ABB RobotStudio station: conveyor SS.rsstn

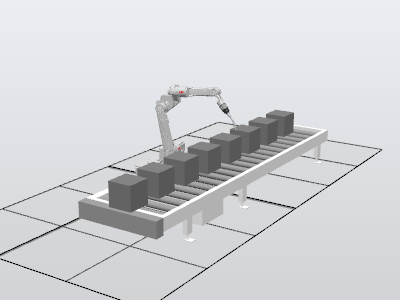
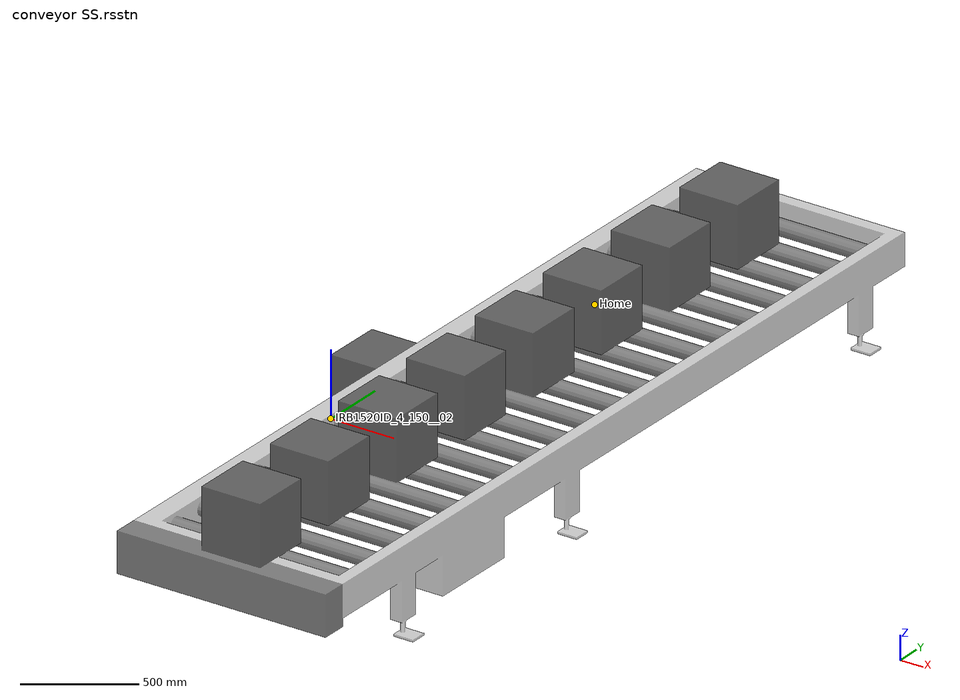
[picture v1: parts stored in the station drawn from their meshes, with robot base, taught points and paths (robot models come from the ABB library and are not in the file)]
Station Station (saved by RobotStudio 22.3.10141.1)
Controller Controller51, task T_ROB1: task frame (RAPID world) sits at (490, 760, 435) mm, rotated rx 0 ry 0 rz -90 deg in the station
Controller Controller51
  mechanical unit ROB_1: IRB1520ID_4_150__02, 6 joints, base frame (760, -490, -435) mm, rotated rx 0 ry 0 rz 90 deg
  mechanical unit CNV1: ?, 1 joints, base frame (0, 0, 0) mm
Layout (positions relative to the parent item):
  - IRB1520ID_4_150__02 [mechanism] at (0, 0, 0) mm; joint values [0.1337, -0.205, 0.1243, -0.1103, 0.9334, 0.1661] (rad or m)
      links: Base, Link1, Link2, Link3, Link4, Link5, Link6
  - Binzel_ID_22 [mechanism, from Tools\Binzel_ID_22.rslib] at (870.51, 99.26, 1138.57) mm, rotated rx 180 ry 41.56 rz 180 deg
  - Conveyor [conveyor]
    - 950_4000_h2 [part] at (1400, -2000, 0) mm, rotated rx 0 ry 0 rz 90 deg, size 4244 x 1170 x 435 mm
    - Box [part], size 300 x 300 x 300 mm
    - ConveyorObject_1 [conveyorobject] at (490, -1725.53, 435) mm, rotated rx 0 ry 0 rz -90 deg
      - Box [part] at (50, 300, 0) mm, size 300 x 300 x 300 mm
    - ConveyorObject_2 [conveyorobject] at (490, -1225.53, 435) mm, rotated rx 0 ry 0 rz -90 deg
      - Box [part] at (50, 300, 0) mm, size 300 x 300 x 300 mm
    - ConveyorObject_3 [conveyorobject] at (490, -725.53, 435) mm, rotated rx 0 ry 0 rz -90 deg
      - Box [part] at (50, 300, 0) mm, size 300 x 300 x 300 mm
    - ConveyorObject_4 [conveyorobject] at (490, -225.53, 435) mm, rotated rx 0 ry 0 rz -90 deg
      - Box [part] at (50, 300, 0) mm, size 300 x 300 x 300 mm
    - ConveyorObject_5 [conveyorobject] at (490, 274.47, 435) mm, rotated rx 0 ry 0 rz -90 deg
      - Box [part] at (50, 300, 0) mm, size 300 x 300 x 300 mm
    - ConveyorObject_6 [conveyorobject] at (490, 774.47, 435) mm, rotated rx 0 ry 0 rz -90 deg
      - Box [part] at (50, 300, 0) mm, size 300 x 300 x 300 mm
    - ConveyorObject_7 [conveyorobject] at (490, 1274.47, 435) mm, rotated rx 0 ry 0 rz -90 deg
      - Box [part] at (50, 300, 0) mm, size 300 x 300 x 300 mm
    - ConveyorObject_8 [conveyorobject] at (490, 1774.47, 435) mm, rotated rx 0 ry 0 rz -90 deg
      - Box [part] at (50, 300, 0) mm, size 300 x 300 x 300 mm
Attachment: Binzel_ID_22 is attached to IRB1520ID_4_150__02 / Link6
Conveyor tracking Connection_4: unit CNV1, TravelOffset=1.3, QueueTrackDistance=0, StartWindowWidth=1.5, SyncSeparation=0, CountsPerMeter=10000
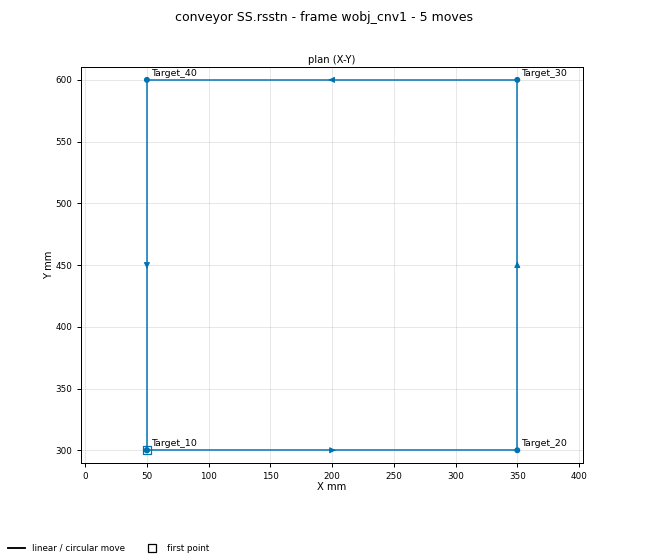
[picture p0: tool path of conveyor SS.rsstn in frame wobj_cnv1, 5 of 7 moves have a stored position in this frame; points joined in program order, loops and branches not executed]
Targets, tools, work objects and paths stored in the station, written as RAPID:
! task T_ROB1
MODULE CalibData
  PERS tooldata tWeldGun:=[TRUE,[[49.841566361,0,372.194826196],[0.981627183,0,0.190808995,0]],[2,[0,0,100],[0,1,0,0],0,0,0]];
  TASK PERS wobjdata wobj_cnv1:=[FALSE,FALSE,"CNV1",[[0,0,0],[1,0,0,0]],[[0,0,0],[1,0,0,0]]];
ENDMODULE

! task T_ROB1
MODULE Module1
  CONST robtarget Home:=[[760,863.614472219,478.738524269],[0.23021145,-0.668582596,0.668582596,0.23021145],[0,-1,0,0],[9E+09,9E+09,9E+09,9E+09,9E+09,0]];
  CONST robtarget Target_10:=[[50,300,300],[0,-0.707106781,0.707106781,0],[0,0,0,0],[9E+09,9E+09,9E+09,9E+09,9E+09,0]];
  CONST robtarget Target_20:=[[350,300,300],[0,-0.707106781,0.707106781,0],[0,0,0,0],[9E+09,9E+09,9E+09,9E+09,9E+09,0]];
  CONST robtarget Target_30:=[[350,600,300],[0,-0.707106781,0.707106781,0],[0,0,0,0],[9E+09,9E+09,9E+09,9E+09,9E+09,0]];
  CONST robtarget Target_40:=[[50,600,300],[0,-0.707106781,0.707106781,0],[0,0,0,0],[9E+09,9E+09,9E+09,9E+09,9E+09,0]];
  CONST robtarget Target_50:=[[50,300,300],[0,-0.707106781,0.707106781,0],[0,0,0,0],[9E+09,9E+09,9E+09,9E+09,9E+09,0]];
  PROC Path_10()
    ActUnit CNV1;
    MoveL Home,v1000,z100,tWeldGun\WObj:=wobj0;
    WaitWObj wobj_cnv1;
    MoveL Target_10,v1000,fine,tWeldGun\WObj:=wobj_cnv1;
    MoveL Target_20,v1000,fine,tWeldGun\WObj:=wobj_cnv1;
    MoveL Target_30,v1000,fine,tWeldGun\WObj:=wobj_cnv1;
    MoveL Target_40,v1000,fine,tWeldGun\WObj:=wobj_cnv1;
    MoveL Target_50,v1000,fine,tWeldGun\WObj:=wobj_cnv1;
    MoveL Home,v1000,z100,tWeldGun\WObj:=wobj0;
    DropWObj wobj_cnv1;
  ENDPROC
ENDMODULE

